// TIA Portal project "5_Assembler" (V19)

(* hardware
DEVICE "S7-1500/ET200MP station_1"  S7-1500 station
   slot 0: "Rail_0"  Rack  6ES7 590-1***0-0AA0
   slot 1: "PLC_1"  CPU 1513-1 PN  6ES7 513-1AL02-0AB0  V2.9
      slot 3: "CPU display_1"  6ES7591-1AA00-0AA0
      slot 32768: "PROFINET interface_1"  X1
         slot 32769: "Port_1"  X1 P1
         slot 32770: "Port_2"  X1 P2
      slot 34817: "Virtual CP interface port_1"  Virtual CP interface port  Virtual CP interface port
*)

// ===== PLC "PLC_1"  CPU 1513-1 PN =====

VAR_GLOBAL   // PLC tag table "Default tag table"
   "Tag_1" AT %M0.1 : Bool;
   "Tag_2" AT %M0.0 : Bool;
   "Tag_3" AT %M0.2 : Bool;
   "Tag_4" AT %M0.3 : Bool;
   "Tag_5" AT %M0.4 : Bool;
   "Tag_6" AT %M0.5 : Bool;
   "Tag_7" AT %M0.6 : Bool;
   "Tag_8" AT %M0.7 : Bool;
   "Tag_9" AT %M1.0 : Bool;
   "Tag_10" AT %M1.1 : Bool;
   "Tag_11" AT %M1.2 : Bool;
   "Tag_12" AT %M1.3 : Bool;
END_VAR

VAR_GLOBAL   // PLC tag table "Tag table from XML_1"
   "Moving X" AT %I0.0 : Bool;
   "Moving Z" AT %I0.1 : Bool;
   "Item detected" AT %I0.2 : Bool;
   "Lid at place" AT %I0.3 : Bool;
   "Lid clamped" AT %I0.4 : Bool;
   "Pos. at limit (lids)" AT %I0.5 : Bool;
   "Base at place" AT %I0.6 : Bool;
   "Base clamped" AT %I0.7 : Bool;
   "Pos. at limit (bases)" AT %I1.0 : Bool;
   "Part leaving" AT %I1.1 : Bool;
   "Start" AT %I1.2 : Bool;
   "Stop" AT %I1.3 : Bool;
   "Auto" AT %I1.4 : Bool;
   "Move X" AT %Q0.0 : Bool;
   "Move Z" AT %Q0.1 : Bool;
   "Grab" AT %Q0.2 : Bool;
   "Lids conveyor" AT %Q0.3 : Bool;
   "Clamp lid" AT %Q0.4 : Bool;
   "Pos. raise (lids)" AT %Q0.5 : Bool;
   "Bases conveyor" AT %Q0.6 : Bool;
   "Clamp base" AT %Q0.7 : Bool;
   "Pos. raise (bases)" AT %Q1.0 : Bool;
   "Start light" AT %Q1.1 : Bool;
   "Stop light" AT %Q1.2 : Bool;
   "Counter" AT %QD30 : DInt;
END_VAR

// folder: System blocks/Program resources

DATA_BLOCK "IEC_Counter_0_DB"   // DB1
{ S7_Optimized_Access := 'TRUE' }
AUTHOR : Simatic
FAMILY : IEC
NAME : CNTR
VERSION : 1.0
// stored: InstanceOfName IEC_COUNTER
"IEC_COUNTER"
BEGIN
END_DATA_BLOCK

DATA_BLOCK "IEC_Timer_0_DB"   // DB2
{ S7_Optimized_Access := 'TRUE' }
AUTHOR : Simatic
FAMILY : IEC
NAME : IEC_TMR
VERSION : 1.0
// stored: InstanceOfName IEC_TIMER
"IEC_TIMER"
BEGIN
END_DATA_BLOCK

DATA_BLOCK "IEC_Timer_0_DB_1"   // DB3
{ S7_Optimized_Access := 'TRUE' }
AUTHOR : Simatic
FAMILY : IEC
NAME : IEC_TMR
VERSION : 1.0
// stored: InstanceOfName IEC_TIMER
"IEC_TIMER"
BEGIN
END_DATA_BLOCK

DATA_BLOCK "IEC_Timer_0_DB_2"   // DB4
{ S7_Optimized_Access := 'TRUE' }
AUTHOR : Simatic
FAMILY : IEC
NAME : IEC_TMR
VERSION : 1.0
// stored: InstanceOfName IEC_TIMER
"IEC_TIMER"
BEGIN
END_DATA_BLOCK

DATA_BLOCK "IEC_Timer_0_DB_3"   // DB5
{ S7_Optimized_Access := 'TRUE' }
AUTHOR : Simatic
FAMILY : IEC
NAME : IEC_TMR
VERSION : 1.0
// stored: InstanceOfName IEC_TIMER
"IEC_TIMER"
BEGIN
END_DATA_BLOCK

// folder: (top level)

ORGANIZATION_BLOCK "Main"   // OB1, LAD, ProgramCycle
TITLE = "Main Program Sweep (Cycle)"
{ S7_Optimized_Access := 'TRUE' }
VERSION : 0.1
   VAR_INPUT
      Initial_Call : Bool;   // Initial call of this OB
      Remanence : Bool;   // =True, if remanent data are available
   END_VAR
   VAR_TEMP   // added for the SCL form of the ladder/FBD networks
      _w1 : Bool;
      _w2 : Bool;
   END_VAR
BEGIN

REGION Network 1: Set the Lid's conveyor
   // The Lid's conveyor will work when in mode auto and press start, or the positioner at the base raise (finish the project). It will stop hwen push the stop button or the lid go through the sensor (On to Off)
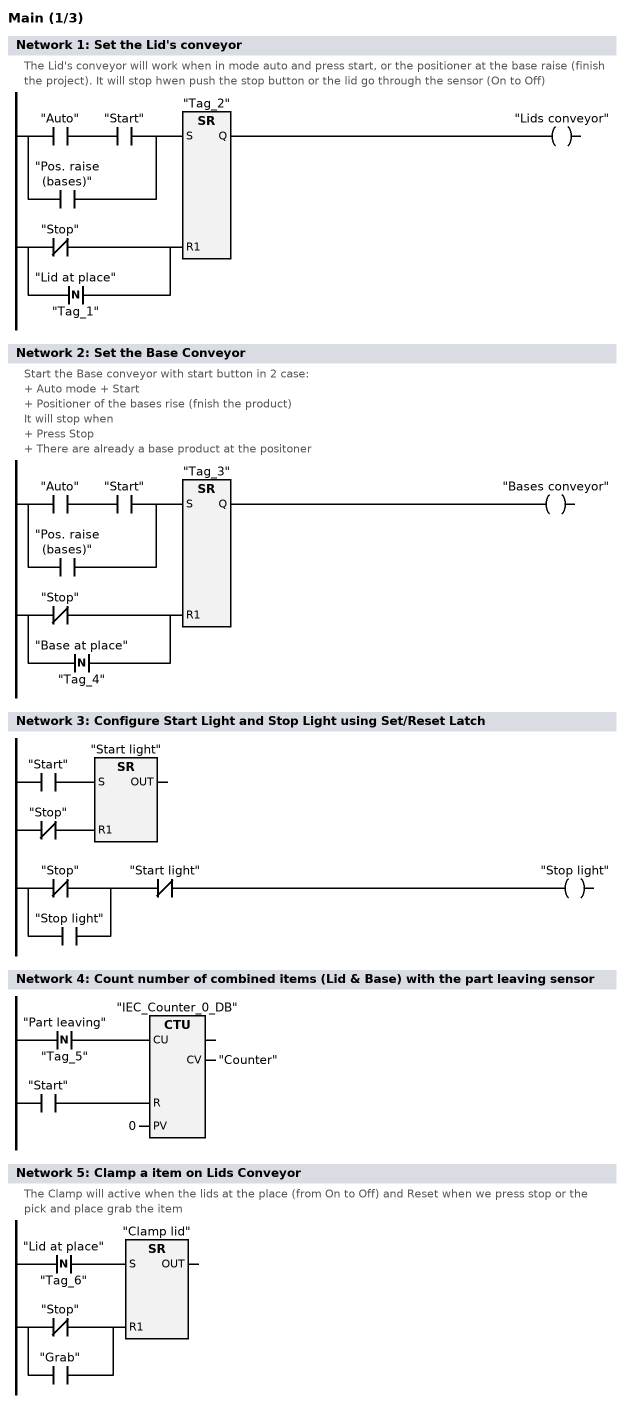
   RUNG wire#powerrail
      Contact( "Auto" )
      Contact( "Start" )
      wire#w1
      S_SR(operand := "Tag_2", r1 := wire#w2)
      Coil( "Lids conveyor" )
   END_RUNG
   RUNG wire#powerrail
      Contact( "Pos. raise (bases)" )
   END_RUNG wire#w1
   RUNG wire#powerrail
      I_Contact( "Stop" )
   END_RUNG wire#w2
   RUNG wire#powerrail
      N_Contact(operand := "Lid at place", bit := "Tag_1")
   END_RUNG wire#w2
   // the same network as SCL:
   #_w1 := NOT "Lid at place" AND "Tag_1";   // falling edge of "Lid at place"
   "Tag_1" := "Lid at place";
   IF ("Auto" AND "Start") OR "Pos. raise (bases)" THEN
       "Tag_2" := TRUE;   // SR flip-flop
   END_IF;
   IF NOT "Stop" OR #_w1 THEN "Tag_2" := FALSE; END_IF;
   "Lids conveyor" := "Tag_2";
END_REGION

REGION Network 2: Set the Base Conveyor
   // Start the Base conveyor with start button in 2 case:
   // + Auto mode + Start
   // + Positioner of the bases rise (fnish the product)
   // It will stop when
   // + Press Stop
   // + There are already a base product at the positoner
   RUNG wire#powerrail
      Contact( "Auto" )
      Contact( "Start" )
      wire#w1
      S_SR(operand := "Tag_3", r1 := wire#w2)
      Coil( "Bases conveyor" )
   END_RUNG
   RUNG wire#powerrail
      Contact( "Pos. raise (bases)" )
   END_RUNG wire#w1
   RUNG wire#powerrail
      I_Contact( "Stop" )
   END_RUNG wire#w2
   RUNG wire#powerrail
      N_Contact(operand := "Base at place", bit := "Tag_4")
   END_RUNG wire#w2
   // the same network as SCL:
   #_w1 := NOT "Base at place" AND "Tag_4";   // falling edge of "Base at place"
   "Tag_4" := "Base at place";
   IF ("Auto" AND "Start") OR "Pos. raise (bases)" THEN
       "Tag_3" := TRUE;   // SR flip-flop
   END_IF;
   IF NOT "Stop" OR #_w1 THEN "Tag_3" := FALSE; END_IF;
   "Bases conveyor" := "Tag_3";
END_REGION

REGION Network 3: Configure Start Light and Stop Light using Set/Reset Latch
   RUNG wire#powerrail
      Contact( "Start" )
      S_SR(operand := "Start light", r1 := wire#w1)
   END_RUNG
   RUNG wire#powerrail
      I_Contact( "Stop" )
   END_RUNG wire#w1
   RUNG wire#powerrail
      I_Contact( "Stop" )
      wire#w2
      I_Contact( "Start light" )
      Coil( "Stop light" )
   END_RUNG
   RUNG wire#powerrail
      Contact( "Stop light" )
   END_RUNG wire#w2
   // the same network as SCL:
   IF "Start" THEN
       "Start light" := TRUE;   // SR flip-flop
   END_IF;
   IF NOT "Stop" THEN "Start light" := FALSE; END_IF;
   "Stop light" := (NOT "Stop" OR "Stop light") AND NOT "Start light";
END_REGION

REGION Network 4: Count number of combined items (Lid & Base) with the part leaving sensor
   #_w1 := NOT "Part leaving" AND "Tag_5";   // falling edge of "Part leaving"
   "Tag_5" := "Part leaving";
   "IEC_Counter_0_DB".CTU(CU := #_w1, R := "Start", PV := 0, CV => "Counter");
END_REGION

REGION Network 5: Clamp a item on Lids Conveyor
   // The Clamp will active when the lids at the place (from On to Off) and Reset when we press stop or the pick and place grab the item
   RUNG wire#powerrail
      N_Contact(operand := "Lid at place", bit := "Tag_6")
      S_SR(operand := "Clamp lid", r1 := wire#w1)
   END_RUNG
   RUNG wire#powerrail
      I_Contact( "Stop" )
   END_RUNG wire#w1
   RUNG wire#powerrail
      Contact( "Grab" )
   END_RUNG wire#w1
   // the same network as SCL:
   #_w1 := NOT "Lid at place" AND "Tag_6";   // falling edge of "Lid at place"
   "Tag_6" := "Lid at place";
   IF #_w1 THEN
       "Clamp lid" := TRUE;   // SR flip-flop
   END_IF;
   IF NOT "Stop" OR "Grab" THEN "Clamp lid" := FALSE; END_IF;
END_REGION

REGION Network 6: Clamp a item on Lids Conveyor
   // The Clamp will active when the bases at the place (from On to Off)
   // Reset when 
   // + we press stop or the pick
   // + The Grab switch from ON to OFF (at the end of the procedure) %This is so smart, love it
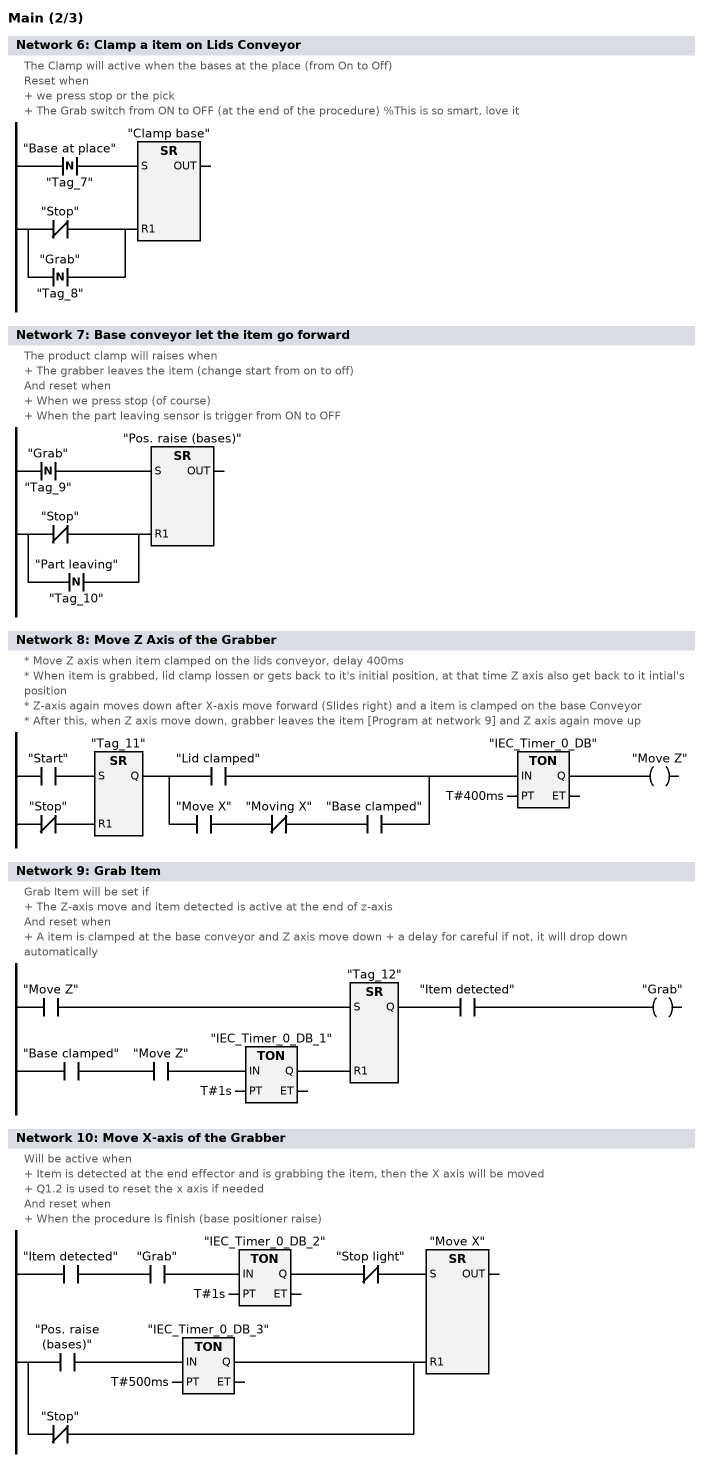
   RUNG wire#powerrail
      N_Contact(operand := "Base at place", bit := "Tag_7")
      S_SR(operand := "Clamp base", r1 := wire#w1)
   END_RUNG
   RUNG wire#powerrail
      I_Contact( "Stop" )
   END_RUNG wire#w1
   RUNG wire#powerrail
      N_Contact(operand := "Grab", bit := "Tag_8")
   END_RUNG wire#w1
   // the same network as SCL:
   #_w1 := NOT "Base at place" AND "Tag_7";   // falling edge of "Base at place"
   "Tag_7" := "Base at place";
   #_w2 := NOT "Grab" AND "Tag_8";   // falling edge of "Grab"
   "Tag_8" := "Grab";
   IF #_w1 THEN
       "Clamp base" := TRUE;   // SR flip-flop
   END_IF;
   IF NOT "Stop" OR #_w2 THEN "Clamp base" := FALSE; END_IF;
END_REGION

REGION Network 7: Base conveyor let the item go forward
   // The product clamp will raises when
   // + The grabber leaves the item (change start from on to off)
   // And reset when
   // + When we press stop (of course)
   // + When the part leaving sensor is trigger from ON to OFF
   RUNG wire#powerrail
      N_Contact(operand := "Grab", bit := "Tag_9")
      S_SR(operand := "Pos. raise (bases)", r1 := wire#w1)
   END_RUNG
   RUNG wire#powerrail
      I_Contact( "Stop" )
   END_RUNG wire#w1
   RUNG wire#powerrail
      N_Contact(operand := "Part leaving", bit := "Tag_10")
   END_RUNG wire#w1
   // the same network as SCL:
   #_w1 := NOT "Grab" AND "Tag_9";   // falling edge of "Grab"
   "Tag_9" := "Grab";
   #_w2 := NOT "Part leaving" AND "Tag_10";   // falling edge of "Part leaving"
   "Tag_10" := "Part leaving";
   IF #_w1 THEN
       "Pos. raise (bases)" := TRUE;   // SR flip-flop
   END_IF;
   IF NOT "Stop" OR #_w2 THEN "Pos. raise (bases)" := FALSE; END_IF;
END_REGION

REGION Network 8: Move Z Axis of the Grabber
   // * Move Z axis when item clamped on the lids conveyor, delay 400ms
   // * When item is grabbed, lid clamp lossen or gets back to it's initial position, at that time Z axis also get back to it intial's position
   // * Z-axis again moves down after X-axis move forward (Slides right) and a item is clamped on the base Conveyor
   // * After this, when Z axis move down, grabber leaves the item [Program at network 9] and Z axis again move up
   IF "Start" THEN
       "Tag_11" := TRUE;   // SR flip-flop
   END_IF;
   IF NOT "Stop" THEN "Tag_11" := FALSE; END_IF;
   "IEC_Timer_0_DB".TON(IN := "Tag_11" AND ("Lid clamped" OR ("Move X" AND NOT "Moving X" AND "Base clamped")),
                        PT := T#400ms);
   "Move Z" := "IEC_Timer_0_DB".Q;
END_REGION

REGION Network 9: Grab Item
   // Grab Item will be set if
   // + The Z-axis move and item detected is active at the end of z-axis
   // And reset when
   // + A item is clamped at the base conveyor and Z axis move down + a delay for careful if not, it will drop down automatically
   "IEC_Timer_0_DB_1".TON(IN := "Base clamped" AND "Move Z", PT := T#1s);
   IF "Move Z" THEN
       "Tag_12" := TRUE;   // SR flip-flop
   END_IF;
   IF "IEC_Timer_0_DB_1".Q THEN "Tag_12" := FALSE; END_IF;
   "Grab" := "Tag_12" AND "Item detected";
END_REGION

REGION Network 10: Move X-axis of the Grabber
   // Will be active when
   // + Item is detected at the end effector and is grabbing the item, then the X axis will be moved
   // + Q1.2 is used to reset the x axis if needed
   // And reset when
   // + When the procedure is finish (base positioner raise)
   "IEC_Timer_0_DB_2".TON(IN := "Item detected" AND "Grab", PT := T#1s);
   "IEC_Timer_0_DB_3".TON(IN := "Pos. raise (bases)", PT := T#500ms);
   IF "IEC_Timer_0_DB_2".Q AND NOT "Stop light" THEN
       "Move X" := TRUE;   // SR flip-flop
   END_IF;
   IF "IEC_Timer_0_DB_3".Q OR NOT "Stop" THEN "Move X" := FALSE; END_IF;
END_REGION

REGION Network 11: Reset the TIMERS
   // We implement this by pressing stop
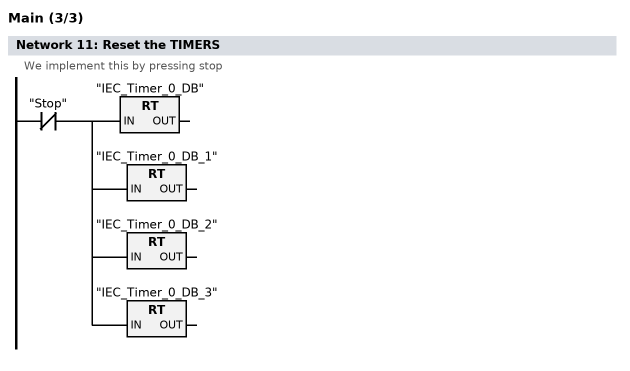
   RUNG wire#powerrail
      I_Contact( "Stop" )
      wire#w1
      RT_Coil( "IEC_Timer_0_DB" )
   END_RUNG
   RUNG wire#w1
      RT_Coil( "IEC_Timer_0_DB_1" )
   END_RUNG
   RUNG wire#w1
      RT_Coil( "IEC_Timer_0_DB_2" )
   END_RUNG
   RUNG wire#w1
      RT_Coil( "IEC_Timer_0_DB_3" )
   END_RUNG
   // the same network as SCL:
   IF NOT "Stop" THEN
       RESET_TIMER("IEC_Timer_0_DB");
       RESET_TIMER("IEC_Timer_0_DB_1");
       RESET_TIMER("IEC_Timer_0_DB_2");
       RESET_TIMER("IEC_Timer_0_DB_3");
   END_IF;
END_REGION
END_ORGANIZATION_BLOCK